(* IEC 61131-3 sources: AXOpen/src/components.siem.identification/ctrl/src/IdentProfile/TypesStructuresAndEnums, 8 files *)

(* ---- eAxo_IID_COMMANDS.st ---- *)
NAMESPACE AXOpen.Components.Siem.Identification
    TYPE PUBLIC
        eAxo_IID_COMMANDS   :   WORD
        (
            eNoCommand		:=  WORD#16#00,
            eRead 			:=  WORD#16#70,
            eWrite			:=  WORD#16#71,
            eReaderStatus 	:=  WORD#16#74,
            eTagStatus 		:=  WORD#16#73,
            eInventory 		:=  WORD#16#69,
            eFormat 		:=  WORD#16#66,
            ePut 			:=  WORD#16#65,
            eWriteID 		:=  WORD#16#67,
            eKillTag 		:=  WORD#16#6A,
            eLockTagBank 	:=  WORD#16#79,
            eEditBlacklist 	:=  WORD#16#7A,
            eGetBlacklist	:=  WORD#16#6C,
            eReadConfig 	:=  WORD#16#61,
            eWriteConfig 	:=  WORD#16#78
        );
    END_TYPE
END_NAMESPACE

(* ---- Axo_IdentDevice_Component_Status.st ---- *)
NAMESPACE AXOpen.Components.Siem.Identification
    {S7.extern=ReadWrite}
    {#ix-attr:[Container(Layout.Stack)]}
    CLASS PUBLIC Axo_IdentDevice_Component_Status  EXTENDS AXOpen.Components.Abstractions.AxoComponent_Status
        VAR PUBLIC
            {#ix-set:AttributeName = "IdentProfile_Status: |[[1]IdentProfileDescription]|"}
            {#ix-attr:[WarningLevel(500)]}
            {#ix-attr:[ErrorLevel(700)]}
            IdentProfile_Status    :   AXOpen.Core.AxoTextList;
        END_VAR
    END_CLASS
END_NAMESPACE

(* ---- Axo_IdentDevice_Config.st ---- *)
NAMESPACE AXOpen.Components.Siem.Identification
    {#ix-attr:[Container(Layout.Stack)]}
    {S7.extern=ReadWrite}
    CLASS PUBLIC Axo_IdentDevice_Config
        VAR PUBLIC
            {#ix-set:AttributeName = "<#Info time#>"}
            InfoTime : LTIME := LT#2S;
            {#ix-set:AttributeName = "<#Error time#>"}
            ErrorTime : LTIME := LT#5S;
            {#ix-set:AttributeName = "<#Start address#>"}
            StartAddress: WORD := WORD#0;
            {#ix-set:AttributeName = "<#Rfid code size#>"}
            RfidCodeSize: WORD := WORD#50;
           {#ix-set:AttributeName = "<#Hardware config data#>"}
            HardwareConfig: AxoByteArray16;
            //:= [BYTE#16#04,BYTE#16#00,BYTE#16#00,BYTE#16#00,BYTE#16#00,BYTE#16#0A,BYTE#16#00,BYTE#16#00,BYTE#16#00,BYTE#16#25,BYTE#16#00,BYTE#16#00,BYTE#16#00,BYTE#16#01,BYTE#16#00,BYTE#16#01]; //default data for RF260R
        END_VAR
    END_CLASS
END_NAMESPACE

(* ---- Axo_IID_IN_EXT_UHF.st ---- *)
NAMESPACE AXOpen.Components.Siem.Identification
    {S7.extern=ReadWrite}
    CLASS Axo_IID_IN_EXT_UHF
        VAR PUBLIC
            LEN_ID                  :   BYTE    :=  BYTE#16#0;     //Length of EPC-ID (0-62)
            MEM_BANK                :   BYTE    :=  BYTE#16#3;     //Memory bank address
            PSWD                    :   DWORD   :=  DWORD#16#0;    //Password
            EDIT_BLACKLIST_MODE     :   BYTE    :=  BYTE#16#0;     //Mode for command "edit blacklist"
            INVENTORY_DURATION      :   WORD    :=  WORD#16#0;     //Duration for command "inventory"
            INVENTORY_DUR_UNIT      :   WORD    :=  WORD#16#0;     //Duration unit for command "inventory"
            LOCK_TAG_BANK_ACTION    :   WORD    :=  WORD#16#0;     //Lock-Action for command "lock-tag-bank"
            LOCK_TAG_BANK_MASK      :   WORD    :=  WORD#16#0;     //Lock Mask for command "lock-tag-bank"
        END_VAR
    END_CLASS
END_NAMESPACE

(* ---- Axo_IID_IN_PN_CONFIGRECORD.st ---- *)
NAMESPACE AXOpen.Components.Siem.Identification
    {S7.extern=ReadWrite}
    CLASS Axo_IID_IN_PN_CONFIGRECORD
        VAR PUBLIC
            nRW         :   WORD;
            nNrAr       :   WORD;
            nApi        :   DWORD;
            nSlot       :   WORD;
            nSubslot    :   WORD;
            record      :   Axo_IID_IN_PN_RECORDDATA ;
        END_VAR
    END_CLASS
END_NAMESPACE

(* ---- Axo_IID_IN_PN_RECORDDATA.st ---- *)
NAMESPACE AXOpen.Components.Siem.Identification
    {S7.extern=ReadWrite}
    CLASS Axo_IID_IN_PN_RECORDDATA
        VAR PUBLIC
            nIndex      :   WORD;
            nLen        :   WORD;
            nTrans      :   WORD;
            nReserve    :   WORD;
            buf         :   ARRAY[0..1034] OF BYTE;
        END_VAR
    END_CLASS
END_NAMESPACE

(* ---- Axo_IID_IN_SYNC.st ---- *)
NAMESPACE AXOpen.Components.Siem.Identification
    {S7.extern=ReadWrite}
    CLASS Axo_IID_IN_SYNC
        VAR PUBLIC
            STATUS_IN_WORK              :   BOOL    :=  FALSE;      //command is in work
            STATUS_INITIALISATION       :   BOOL    :=  FALSE;      //initialisation is in work
            STATUS_LAST_CMD_INIT        :   BOOL    :=  FALSE;      //flag for initialisation
            sreset_request              :   BOOL    :=  FALSE;      //show that one app is in sreset
            acyc_active                 :   BOOL    :=  FALSE;      //acyc service is running
            reset_request               :   BOOL    :=  FALSE;      //shows that one reset-instruction is wait for ends of acyclic commands
            AC_H                        :   BOOL    :=  FALSE;      //ack counter high
            AC_L                        :   BOOL    :=  FALSE;      //ack counter low
            CC_H                        :   BOOL    :=  FALSE;      //cmd counter high
            CC_L                        :   BOOL    :=  FALSE;      //cmd counter low
            old_CC_H                    :   BOOL    :=  FALSE;      //previous ack counter high
            old_CC_L                    :   BOOL    :=  FALSE;      //previous ack counter low
            old_AC_H                    :   BOOL    :=  FALSE;      //previous cmd counter high
            old_AC_L                    :   BOOL    :=  FALSE;      //previous cmd counter low
            cyc_control                 :   WORD    :=  WORD#16#0;  //cyclic control word
            cyc_status                  :   WORD    :=  WORD#16#0;  //cyclic status word
            SRESET_active               :   BOOL    :=  FALSE;      //sreset active bit (cyc status word)
            SRESET_cyc                  :   BOOL    :=  FALSE;      //sreset control bit (cyc control word)
            RPTCMD_cyc                  :   BOOL    :=  FALSE;      //repeat control bit (cyc control word)
            RPTCMD_active               :   BOOL    :=  FALSE;      //repeat active bit (cyc status word)
            INIT_cyc                    :   BOOL    :=  FALSE;      //init control bit (cyc control word)
            init_active                 :   BOOL    :=  FALSE;      //init status bit (cyc status word)
            presence                    :   BOOL    :=  FALSE;      //presence-bit
            buf_header                  :   UINT    :=  UINT#11;    //length pib-header
            sequence_number             :   UINT    :=  UINT#0;     //sequence number (pib-header)
            config_value                :   BYTE    :=  BYTE#16#4;  //config mode for pdu-detection
            offset                      :   UINT    :=  UINT#0;     //offset for cyclic status/control word
            index                       :   UINT    :=  UINT#0;     //index for WRREC/RDREC
            buf_max                     :   UINT    :=  UINT#240;   //acyclic datagram buffer size
            instruction_set             :   BOOL    :=  FALSE;      //state for instruction set (1=RF68xR; 0=old CMs)
            index_set                   :   BOOL    :=  TRUE;       //state for DS-index (1=PROFINET; 0=PROFIBUS)
            timeout_repeat              :   TIME    :=  T#5S;       //timeout for repeat
            timeout_reset               :   TIME    :=  T#1M;       //timeout for init
            state                       :   UINT    :=  UINT#0;     //variable for statemachine
            buf_maxdata                 :   UINT    :=  UINT#229;   //user data size
            pnConfigRecord              :   Axo_IID_IN_PN_CONFIGRECORD;
        END_VAR
    END_CLASS
END_NAMESPACE

(* ---- AxoByteArray16.st ---- *)
NAMESPACE AXOpen.Components.Siem.Identification
    {S7.extern=ReadWrite}
    CLASS PUBLIC AxoByteArray16 EXTENDS AXOpen.Core.AxoByteArray
        VAR PUBLIC
            Data : ARRAY [0..15] OF BYTE;
        END_VAR
    END_CLASS
END_NAMESPACE
